FUNCTION_BLOCK FB_HaltNC_TestDouble IMPLEMENTS  I_Halt
VAR
    bError : BOOL;
    nErrorID : UDINT := 19000;
END_VAR

PROPERTY Aborted : BOOL
GET
END_GET
END_PROPERTY

PROPERTY Active : BOOL
GET
Active := TRUE;
END_GET
END_PROPERTY

PROPERTY Busy : BOOL
GET
END_GET
END_PROPERTY

METHOD ClearStatus
END_METHOD

PROPERTY CommandHalt : BOOL
SET
END_SET
END_PROPERTY

PROPERTY Done : BOOL
GET
END_GET
END_PROPERTY

PROPERTY Error : BOOL
GET
Error := bError;
END_GET
SET
bError := Error;
END_SET
END_PROPERTY

PROPERTY ErrorID : UDINT
GET
ErrorId := nErrorID;
END_GET
SET
nErrorId := ErrorID;
END_SET
END_PROPERTY

METHOD Halt
VAR_INPUT
    Deceleration	: LREAL := 0;
    Jerk	: LREAL := 0;
    BufferMode	: MC_BufferMode := MC_BufferMode.MC_Aborting;
END_VAR
END_METHOD

PROPERTY Message : T_MAXSTRING
GET
END_GET
END_PROPERTY

END_FUNCTION_BLOCK

(* stored: Version 1.1.0.1
   POU FB_HaltNC_TestDouble: Id {f9b66d85-7bb4-402b-9f8b-2a0adea12002}, SpecialFunc None
   Property Aborted: Id {dcd96d02-fc41-4439-b399-ffb9de51b6a6}
   Get Get: Id {32ea644c-2297-41d5-9c0f-de4abdcc0a05}
   Property Active: Id {de01ada0-e7f0-48bc-bf66-59fd6b84f4d5}
   Get Get: Id {ff6da14b-65c4-4946-baa0-2f64630851e4}
   Property Busy: Id {ecfea804-16ec-4572-9424-25e12b445ee2}
   Get Get: Id {9a7dce4c-e6a4-4f0c-bf86-cb8f0d6de522}
   Method ClearStatus: Id {926c075d-bb71-43bb-b2c3-d039de87d848}
   Property CommandHalt: Id {5a4d8f78-05a5-40fb-b10c-445da57e98d8}
   Set Set: Id {7618836d-62fb-4a17-b12d-c39950d5a82b}
   Property Done: Id {f35d2583-5ac2-46cb-8465-dc7b5f25ec3f}
   Get Get: Id {a79b7878-9f49-4fbd-9504-8b8936b04073}
   Property Error: Id {f52da4d2-0b9a-4928-b781-7a19d609abc5}
   Get Get: Id {6ccd1c8c-a7f2-460f-aed1-6737e0b752a8}
   Set Set: Id {548bb34b-cf95-4acf-b5c1-a3527f630e39}
   Property ErrorID: Id {61771d5f-635c-4dcf-96b8-37aff8730699}
   Get Get: Id {6997e5ed-2ca0-4ccd-adc8-426dab1bad9c}
   Set Set: Id {ba886be4-928a-4dcc-ab5b-bfa33d22eae1}
   Method Halt: Id {2294bac2-3031-41ca-9141-34b574671001}
   Property Message: Id {98d02838-f1f1-467b-9553-0611cc90df48}
   Get Get: Id {5fb5cb0f-5bfd-4fe1-aaf1-0e72d32ad429} *)
